PROGRAM MAIN
VAR
    sensorA, sensorB, motorLinksDraaiend, motorRechtsDraaiend, alarm: BOOL;
    fbFlankSensorA, fbFlankSensorB: R_TRIG; // Rising edge detection for sensors
END_VAR

(*
Draairichting van een motor (2 regel code)

Op de as van een motor worden twee sensoren gemonteerd bv reflex fotocellen.
Bepaal de draairichting met flankdetectie.


Uitbreiding: Om een verplaatsbare pomp niet te beschadigen mag een elektrische motor enkel links draaien. 
Daarom wordt de draairichting gedetecteerd door middel van vorige oefening. 
Wanneer de motor links aanloopt is er normale werking.
Als de motor rechts aanloopt zal hij onmiddellijk stilvallen en een rood alarmlicht zal branden.
*)

fbFlankSensorA(CLK:=sensorA); fbFlankSensorB(CLK:=sensorB);
motorLinksDraaiend := fbFlankSensorA.Q AND NOT sensorB; 
motorRechtsDraaiend := fbFlankSensorB.Q AND NOT sensorA;



// Uitbreiding
alarm := NOT motorLinksDraaiend;

END_PROGRAM

(* stored: Version 1.1.0.1, ProductVersion 3.1.4024.12
   POU MAIN: Id {37994f21-3bc5-4ef9-8a99-b480fc2c96cd}, SpecialFunc None *)
